Staubli VAL3: start.pgx

program start()
  local num l_nSioCtrl
begin
  bInputBuffering=true
  sInputBuffering="subscriber"
  bTaskManager=true
  cls()
  resetMotion()
  userPage()
  l_nSioCtrl=sioCtrl(siConn,"timeout",5)
  if (l_nSioCtrl<0)
    putln("Could not set the timeout")
  endIf
  putln("Starting task")
  l_nSioCtrl=sioCtrl(soConn,"timeout",5)
  if (l_nSioCtrl<0)
    putln("Could not set the timeout")
  endIf
  taskCreate sInputBuffering,50,SIMPLE_MSG(trajMsg:prefix.nLength,trajMsg:header.nMsgType)
  taskCreate "t_manage",10,TASK_MANAGER()
end
